INTERFACE I_XP_Track  EXTENDS I_CH_Object

METHOD AddMover : HRESULT
VAR_INPUT
	ipMover : I_XP_Mover;
END_VAR
END_METHOD

METHOD AddToGroup : HRESULT
VAR_INPUT
	iGroup : I_XP_Group;
END_VAR
END_METHOD

{attribute 'monitoring':='call'}
PROPERTY ClosedLoop : BOOL
GET
END_GET
END_PROPERTY

METHOD Configure : HRESULT
VAR_INPUT
END_VAR
END_METHOD

METHOD Configuring : HRESULT
VAR_INPUT
END_VAR
END_METHOD

{attribute 'monitoring':='call'}
PROPERTY CtsMoversOnTrack : UINT
GET
END_GET
END_PROPERTY

METHOD Disable : HRESULT
VAR_INPUT
END_VAR
END_METHOD

METHOD Enable : HRESULT
VAR_INPUT
END_VAR
END_METHOD

{attribute 'monitoring':='call'}
PROPERTY Feedback : I_XP_Feedback
GET
END_GET
END_PROPERTY

(* Calculates which gap the mover should have on a position
	The gap results from the last station crossed.
	If several stations are possible ( switch), the largest gap is displayed here *)
METHOD GapAtPosition : LREAL
VAR_INPUT
	fPosOnTrack : LREAL;//[mm]	
END_VAR
END_METHOD

{attribute 'monitoring':='call'}
//[mm]
PROPERTY Length : LREAL
GET
END_GET
END_PROPERTY

{attribute 'monitoring':='call'}
PROPERTY PlanarTrack : REFERENCE TO MC_PlanarTrack
GET
END_GET
END_PROPERTY

METHOD RemoveFromGroup : HRESULT
END_METHOD

METHOD Reset : HRESULT
VAR_INPUT
END_VAR
END_METHOD

(* Returns the first station on current track who has exact thsi position or is ahead
	If no station on this track, result is maybe on another track*)
METHOD StationAhedPosition : I_XP_Station
VAR_INPUT
	fPosOnTrack : LREAL;//[mm]	
END_VAR
END_METHOD

{attribute 'monitoring':='call'}
//List of interfaces to stations on this track
PROPERTY StationsOnTrack : I_CH_List
GET
END_GET
END_PROPERTY

{attribute 'monitoring':='call'}
//List of interfaces from other tracks
PROPERTY TracksAhead : I_CH_List
GET
END_GET
END_PROPERTY

{attribute 'monitoring':='call'}
//List of interfaces from other tracks
PROPERTY TracksBehinde : I_CH_List
GET
END_GET
END_PROPERTY

{attribute 'monitoring':='call'}
PROPERTY TracksEndAtThis : REFERENCE TO  ARRAY[0..(XPlanarParameterlist.N_MAX_STATIONS_AHEAD_OR_BEHIND-1)] OF I_XP_Track
GET
END_GET
END_PROPERTY

{attribute 'monitoring':='call'}
PROPERTY TracksStartFromThis : REFERENCE TO ARRAY[0..(XPlanarParameterlist.N_MAX_STATIONS_AHEAD_OR_BEHIND-1)] OF I_XP_Track
GET
END_GET
END_PROPERTY

END_INTERFACE

(* stored: Version 1.1.0.1, ProductVersion 3.1.4024.12
   Itf I_XP_Track: Id {3432d48a-a726-4b83-a12f-d272099ac173}
   Method AddMover: Id {2b200b3a-86da-49d6-8e5e-103f557e3dc0}
   Method AddToGroup: Id {302bb858-5b9c-468d-9362-6205f917332d}
   Property ClosedLoop: Id {a2468070-3b2b-421b-9055-75836b9066dd}
   Get Get: Id {af83d3fa-3fcc-4aee-8d0c-95c02d967deb}
   Method Configure: Id {c62dbb08-9afd-4532-97d6-aa5d2b5a1ef8}
   Method Configuring: Id {99ddac7c-0893-4b9e-849d-6ec656e69701}
   Property CtsMoversOnTrack: Id {11733006-6736-4805-a3ef-77a950d4f32e}
   Get Get: Id {15f0dbd1-68cd-4f2a-8369-848e0f2a1464}
   Method Disable: Id {846f7e23-ca61-4e09-aaee-8a11a2364d2a}
   Method Enable: Id {1d1eefd1-801d-44e6-af56-039a1cf4679d}
   Property Feedback: Id {04374df7-b187-4c05-b1de-93763caf4aa2}
   Get Get: Id {0b605435-87de-4ddb-b3ce-157455508880}
   Method GapAtPosition: Id {4387fda7-8415-4e9f-ab5a-c5b1be5d697b}
   Property Length: Id {35044908-1b9c-4871-a3ff-14ae54040ef3}
   Get Get: Id {3d6b015c-79c3-4572-a415-52ab650d4cd2}
   Property PlanarTrack: Id {54d6428b-7468-4a87-b287-ed624feebdbb}
   Get Get: Id {4b4abc4a-0f9b-46c5-ab81-216b9e4230d2}
   Method RemoveFromGroup: Id {5404cd47-f9b8-4221-b66c-c23d46a77129}
   Method Reset: Id {2f8c91d6-0cfd-4177-bb04-2e49e3ecd0de}
   Method StationAhedPosition: Id {8f31d0eb-b127-41f6-a9ea-ceefd386b8d6}
   Property StationsOnTrack: Id {e9fcb1ff-197a-4c9e-9a9a-8b0acd76a517}
   Get Get: Id {35065c9a-f7a7-4fd2-bbc2-b5f6d10156cd}
   Property TracksAhead: Id {01ae3317-26a9-4790-a3fe-0dfe598d8739}
   Get Get: Id {a77fe1ec-8bd8-482c-afed-45600b1a59cb}
   Property TracksBehinde: Id {63639ca9-73ad-4626-b3c9-81144942761a}
   Get Get: Id {688effa3-acac-48c2-9e99-dda83a78d8df}
   Property TracksEndAtThis: Id {2b7d0403-8812-431a-92f0-60cef6f1780d}
   Get Get: Id {8cf88d14-2cf5-4374-a40a-bda85ffb07df}
   Property TracksStartFromThis: Id {96711d99-9b22-4448-8ae5-5143ac7d8434}
   Get Get: Id {7ea3e3f5-20d0-47aa-b1b0-ea4b617cfbd1} *)
